{attribute 'qualified_only'}
VAR_GLOBAL
	bAxisError	: BOOL;
END_VAR

(* stored: Version 1.1.0.1, ProductVersion 3.1.4020.6
   GVL GVL: Id {69b728e0-95ed-4afd-b0b6-7ddd4df649cc} *)
